(* IEC 61131-3 sources: inproshop/test7_exported/OP11/2.PRG, 9 files *)

(* ---- OP11_Communication.st ---- *)
PROGRAM OP11_Communication
VAR
	HeartdelayON:TON;
	HeartdelayOFF:TON;
	MasterHeartdelayON:TON;
	MasterHeartdelayOFF:TON;
END_VAR

//心跳输出
IF CPU_Clock.Clock_1s THEN
	DB1105_Communication.TO_OPXX.Heart:=1;
ELSE
	DB1105_Communication.TO_OPXX.Heart:=0;
END_IF
//给前站安全信号
IF TRUE THEN
	DB1105_Communication.TO_OPXX.Safe:=1;
ELSE
	DB1105_Communication.TO_OPXX.Safe:=0;
END_IF;

HeartdelayON(IN:= DB1105_Communication.From_OPXX.Heart=1, PT:= T#2S, Q=> , ET=> );
HeartdelayOFF(IN:= DB1105_Communication.From_OPXX.Heart=0, PT:= T#2S, Q=> , ET=> );
//前站掉线报警
IF (HeartdelayON.Q OR HeartdelayOFF.Q) AND NOT DB1100_Control.Mode.Status.OfflineMode  THEN
	DB1170_Fault.Stop.BeforStation_Communication_Rrror:=TRUE;
END_IF

//主站心跳通讯检测
MasterHeartdelayON(IN:= DB1105_Communication.FromMaster.Heart=1, PT:= T#2S, Q=> , ET=> );
MasterHeartdelayOFF(IN:= DB1105_Communication.FromMaster.Heart=0, PT:= T#2S, Q=> , ET=> );
//主站掉线报警
IF (MasterHeartdelayON.Q OR MasterHeartdelayOFF.Q) AND NOT DB1100_Control.Mode.Status.OfflineMode  THEN
	DB1170_Fault.Stop.MasterTimeOut:=TRUE;
END_IF

//与主站配方不一致报警
IF DB1105_Communication.FromMaster.MasterRecipeID<>DB1102_Recipe.RecipeNum AND NOT DB1100_Control.Mode.Status.OfflineMode THEN
	DB1170_Fault.Stop.MaterReipeDiscrepancy:=TRUE;
END_IF

(* ---- OP11_Control.st ---- *)
PROGRAM OP11_Control
VAR
	FB_ModeControl_instance:FB_ModeControl_V1;
	FB_Count_instance:ARRAY[0..2] OF FB_Count;
END_VAR

(**********模式切换功能***********)
FB_ModeControl_instance(
	iClock:= CPU_Clock,
	iStartDelay:= T#100MS,
	iEstop:=DB1170_Fault.EstopTotal,
	iAlam:=DB1170_Fault.StopTotal,
	iWarn:=DB1170_Fault.RunTotal,
	ioMachine:= DB1100_Control.Machine,
	ioMode:=DB1100_Control.Mode);

(********************计数****************************)
//总计数
FB_Count_instance[0](
	ioCount:= DB1103_Count.Total,
	iClock:= CPU_Clock,
	iDayStartTime:= CPU_Clock.DayStartTime,
	iNightStartTime:=CPU_Clock.NightStartTime);

//OK计数
FB_Count_instance[1](
	ioCount:= DB1103_Count.OK,
	iClock:= CPU_Clock,
	iDayStartTime:= CPU_Clock.DayStartTime,
	iNightStartTime:=CPU_Clock.NightStartTime);

//NG计数
FB_Count_instance[2](
	ioCount:= DB1103_Count.NG,
	iClock:= CPU_Clock,
	iDayStartTime:= CPU_Clock.DayStartTime,
	iNightStartTime:=CPU_Clock.NightStartTime);

(***********良率计算***********)
//良率统计
IF DB1103_Count.Total.Today.Total<>0 THEN
	DB1103_Count.Yield:=DB1103_Count.OK.Today.Total/DB1103_Count.Total.Today.Total;
ELSE
	DB1103_Count.Yield:=0;
END_IF
//良率清零
IF DB1103_Count.Clear THEN
	DB1103_Count.Total.Today.Total:=0;
	DB1103_Count.OK.Today.Total:=0;
	DB1103_Count.NG.Today.Total:=0;
	DB1103_Count.Clear:=FALSE;
END_IF

(********程序调用*******)
OP11_DI_Mirror();
OP11_Communication();
OP11_Recipe();
OP11_Graph();
OP11_DriveControl();
OP11_DO_Mirror();
OP11_Fault();
OP11_Other();

(* ---- OP11_DI_Mirror.st ---- *)
PROGRAM OP11_DI_Mirror
VAR
	i:INT;//循环用变量
	Page:INT;
	Monitor:ARRAY[0..15] OF Str_IOMonitor;
	Status:WORD;
	Map:BOOL;
END_VAR

ACT_MAP();
ACT_Comment();
ACT_Status();

(* ---- OP11_DO_Mirror.st ---- *)
PROGRAM OP11_DO_Mirror
VAR
	i:INT;//循环用变量
	Page:INT;
	Monitor:ARRAY[0..15] OF Str_IOMonitor;
	Status:WORD;
	Map:BOOL;
	Startlamp1:BOOL;
	Startlamp2:BOOL;
END_VAR

ACT_MAP();
ACT_Comment();
ACT_Status();

(* ---- OP11_DriveControl.st ---- *)
PROGRAM OP11_DriveControl
VAR
	FB_Cylinder_instance :ARRAY[0..63]OF FB_Cylinder_V1;
	FB_Vacuum_instance :ARRAY[0..31]OF FB_Vacuum_V1;
	FB_Axis_Instance:ARRAY[0..31]OF FB_Axis_V1_3;
	FB_Sensor_instance :ARRAY[0..200]OF FB_Sensor_V1_1;
	FB_TcpClient_Instance:ARRAY[0..31]OF FB_TcpClient;
	FB_DoubleStart_Instance:ARRAY[1..4]OF FB_DoubleStart;
	FB_Epson_V1_Instance:ARRAY[1..1]OF FB_Epson_V1;
	FB_Kuka_V1_Instance:ARRAY[1..2]OF FB_Kuka6_V1;
	FB_Rotdisk_V1_Instance:ARRAY[1..1]OF FB_Rotdisk_V1;
	FB_Stopper_V1_Instance:ARRAY[1..1]OF FB_Stopper_V1;
	FB_Motor_Instance:ARRAY[1..1]OF FB_Motor;
	FB_Heating_Instance:ARRAY[1..1]OF FB_Heating;
	FB_Gear_Instance:ARRAY[1..1]OF FB_Gear;
	FB_AAS_Instance:ARRAY[1..1]OF FB_AAS;
	FB_AirLeak_Instance:ARRAY[1..2]OF FB_AirLeak;
	FB_Palletizing_Instance:ARRAY[1..3]OF FB_Palletizing;
END_VAR
VAR
	i:INT;//循环变量用
	j:INT;//循环变量用
END_VAR

VAR
	TempKUKA1InPut AT %IB4500:ARRAY[0..63]OF BYTE;
	TempKUKA1OutPut AT %QB4500:ARRAY[0..63]OF BYTE;
	TempKUKA2InPut AT %IB4600:ARRAY[0..63]OF BYTE;
	TempKUKA2OutPut AT %QB4600:ARRAY[0..63]OF BYTE;
END_VAR
VAR
	PowerLimitDelay:ARRAY[0..16] OF TON;//超出额定电流
END_VAR

ACT_Axis();
ACT_Cylinder();
ACT_Vacuum();
ACT_Epson();
ACT_Kuka();
ACT_Sensor();
ACT_Motor();
ACT_Rotdisk();
ACT_AI();
ACT_Stopper();

ACT_Pallet();

(* ---- OP11_Fault.st ---- *)
PROGRAM OP11_Fault
VAR
	i:UINT;//循环变量用
	Pobool_IN: POINTER TO BOOL;//输入报警指针地址获取；
	Pobool_OUT: POINTER TO BOOL;//输出报警指针地址获取；
	EstopMAP:ARRAY[0..255] OF BOOL;
	StopMAP:ARRAY[0..999] OF BOOL;
	RunMAP:ARRAY[0..255] OF BOOL;
	Size:UINT;//数组数量
	Estop_R:R_TRIG;//急停上升沿
	Stop_R:R_TRIG;//暂停上升沿
	Run_R:R_TRIG;//警告上升沿
	StopFaultDelay:ARRAY[1..10]OF TON;//停止报警延时
END_VAR

//气缸报警地址映射
SizeOfAry(In:=DB1150_DriveControl.CylCtrl,Out=>Size);
FOR i:=0 TO Size-1 BY 1 DO
	DB1170_Fault.Stop.Cyl[I]:=DB1150_DriveControl.CylCtrl[i].Status.Error;
END_FOR
//真空报警映射
SizeOfAry(In:=DB1150_DriveControl.VacCtrl,Out=>Size);
FOR i:=0 TO Size-1 BY 1 DO
	DB1170_Fault.Stop.Vac[I]:=DB1150_DriveControl.VacCtrl[i].Status.Error;
END_FOR
//轴报警映射
SizeOfAry(In:=DB1150_DriveControl.AxisCtrl,Out=>Size);
FOR i:=0 TO Size-1 BY 1 DO
	DB1170_Fault.Stop.Axis[I]:=DB1150_DriveControl.AxisCtrl[i].Status.Error;
END_FOR

//急停报警
DB1170_Fault.Estop.EstopButton:=NOT DB1100_Control.Machine.EmgSafetyRelay;

//暂停故障

DB1170_Fault.Stop.SafeDoorOpen:=NOT DB1100_Control.Machine.SafetyDoorRelay;

//提示

ACT_MAP();
ACT_HMI_Jump();

(* ---- OP11_Graph.st ---- *)
PROGRAM OP11_Graph
VAR
	IntitalTimeDelay:ARRAY[1..9,0..10] OF TON;//初始化流程用
	AutoTimeDelay:ARRAY[1..9,0..10] OF TON;//自动流程用

	Init:ARRAY[1..20]OF Str_Graph := [20((Complete := TRUE))];//初始化
	Auto:ARRAY[1..20]OF Str_Graph;//自动
	Start:ARRAY[1..9] OF BOOL;//自动启动条件
	i:INT;//循环变量用

	AgingPutAllowNo:INT;//老化允许放编号
	AgingPickAllowNo:INT;//老化允许取编号
	BufferPutAllowNo:INT;//缓存台允许放编号

	AgingPutAllow:BOOL;//老化允许放
	AgingPickAllow:BOOL;//老化允许取
	BufferPutAllow:BOOL;//缓存台允许放

	BufferPickAllow:BOOL;//缓存台允许取
	TestPickAllow:BOOL;//测试台允许取
	TestPutAllow:BOOL;//测试台允许放
	PalletProductPutAllow:BOOL;//码垛区域允许放产品
	PalletPartitionPutAllow:BOOL;//码垛区域允许放隔板
	PalletPartitionPickAllow:BOOL;//码垛区域允许取隔板
	NgPutAllow:BOOL;//NG区域允许放料

	BufferPickAllowNo:INT;//缓存台允许取编号
	TestPickAllowNo:INT;//测试台允许取编号
	TestPutAllowNo:INT;//测试台允许放编号
	PalletProductPutAllowNo:INT;//码垛区域允许放产品编号
	PalletPartitionPutAllowNo:INT;//码垛区域允许放隔板编号

	PartitionInRobot:BOOL;//机械手上有隔板

	X1Point:INT;//X1轴
	X2Point:INT;//X1轴
	BufferDisable:ARRAY[0..4]OF BOOL;

END_VAR

ACT_InitST1();
ACT_InitST2();
ACT_InitST3();
ACT_InitST4();
ACT_InitST5();
ACT_InitST6();

ACT_AutoRunST1_气密1测试();
ACT_AutoRunST2_气密2测试();
ACT_AutoRunST3_气密3测试();
ACT_AutoRunST4_气密4测试();
ACT_AutoRunST5_上料机械手();
ACT_AutoRunST6_码垛机械手();

(* ---- OP11_Other.st ---- *)
PROGRAM OP11_Other
VAR
	i:INT;//循环变量
	MaterialCode: INT;
END_VAR

(* ---- OP11_Recipe.st ---- *)
PROGRAM OP11_Recipe
VAR
	i:INT;
	DownLoad_R:R_TRIG;
	Download_F:F_TRIG;
	Change:R_TRIG;
END_VAR
VAR RETAIN PERSISTENT
	RecipeNum AT %MB131074 : INT;
END_VAR

//主站一键切换配方
IF To_Slave.OnLineMode=1 THEN
	IF DB1102_Recipe.DownLoad THEN
		To_Slave.RecipeDownLoad:=1;
	ELSE
		To_Slave.RecipeDownLoad:=0;
	END_IF
	To_Slave.RecipeID:=DB1102_Recipe.RecipeNumTemp;
ELSE
	To_Slave.RecipeDownLoad:=0;
END_IF

//配方名
DB1102_Recipe.RecipeName:=DB1102_Recipe.TypeData[DB1102_Recipe.RecipeNum].Name;

//配方参数修改使能
IF DB1102_Recipe.RecipeNum=DB1102_Recipe.RecipeNumTemp THEN
	DB1102_Recipe.ParameterChangePmt:=TRUE;
ELSE
	DB1102_Recipe.ParameterChangePmt:=FALSE;
END_IF

//配方允许切换使能
DB1102_Recipe.RecipeChangePmt:=DB1100_Control.Mode.Status.ManualMode ;

//配方提取
DB1102_Recipe.TypeDataCur:=DB1102_Recipe.TypeData[DB1102_Recipe.RecipeNum];

IF RecipeNum<>DB1102_Recipe.RecipeNumTemp THEN
	DB1102_Recipe.RecipeNameTemp:=DB1102_Recipe.TypeData[DB1102_Recipe.RecipeNumTemp].Name;
	RecipeNum:=DB1102_Recipe.RecipeNumTemp;
END_IF

DownLoad_R(CLK:= DB1102_Recipe.DownLoad);
DownLoad_F(CLK:= DB1102_Recipe.DownLoad);
ACT_Download();
ACT_Upload();
